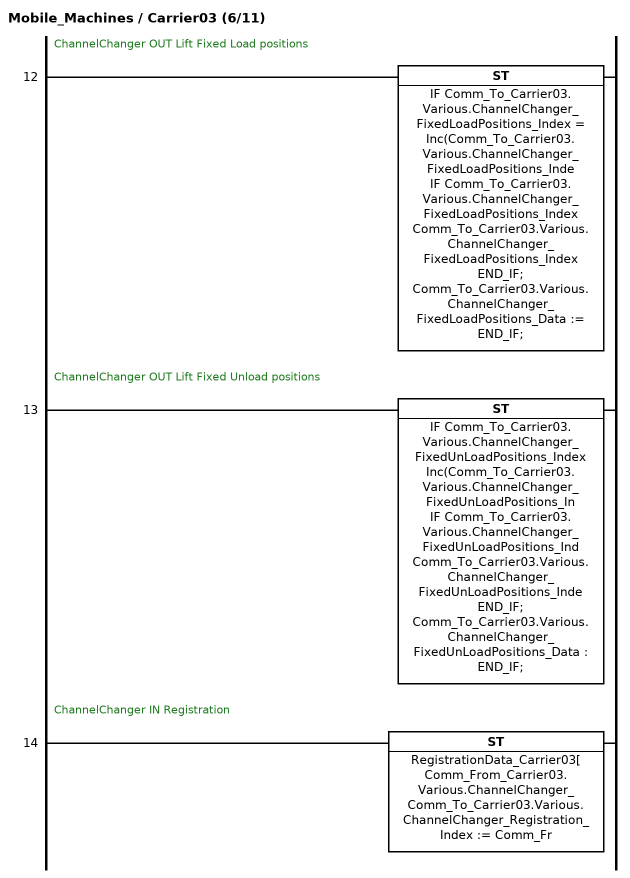
(* [picture p54: Mobile_Machines / Carrier03, rungs 12-14] *)
(* Rung 12: ChannelChanger OUT Lift Fixed Load positions *)
IF Comm_To_Carrier03.Various.ChannelChanger_FixedLoadPositions_Index = Comm_From_Carrier03.Various.ChannelChanger_FixedLoadPositions_Index THEN
	Inc(Comm_To_Carrier03.Various.ChannelChanger_FixedLoadPositions_Index);
	IF Comm_To_Carrier03.Various.ChannelChanger_FixedLoadPositions_Index > 199 THEN
		Comm_To_Carrier03.Various.ChannelChanger_FixedLoadPositions_Index := 0;
	END_IF;
	Comm_To_Carrier03.Various.ChannelChanger_FixedLoadPositions_Data := FixedLoadPosition_Array[Comm_To_Carrier03.Various.ChannelChanger_FixedLoadPositions_Index];
END_IF;
(* Rung 13: ChannelChanger OUT Lift Fixed Unload positions *)
IF Comm_To_Carrier03.Various.ChannelChanger_FixedUnLoadPositions_Index = Comm_From_Carrier03.Various.ChannelChanger_FixedUnLoadPositions_Index THEN
	Inc(Comm_To_Carrier03.Various.ChannelChanger_FixedUnLoadPositions_Index);
	IF Comm_To_Carrier03.Various.ChannelChanger_FixedUnLoadPositions_Index > 199 THEN
		Comm_To_Carrier03.Various.ChannelChanger_FixedUnLoadPositions_Index := 0;
	END_IF;
	Comm_To_Carrier03.Various.ChannelChanger_FixedUnLoadPositions_Data := FixedUnloadPosition_Array[Comm_To_Carrier03.Various.ChannelChanger_FixedUnLoadPositions_Index];
END_IF;
(* Rung 14: ChannelChanger IN Registration *)
RegistrationData_Carrier03[Comm_From_Carrier03.Various.ChannelChanger_Registration_Index] := Comm_From_Carrier03.Various.ChannelChanger_Registration_Data;
Comm_To_Carrier03.Various.ChannelChanger_Registration_Index := Comm_From_Carrier03.Various.ChannelChanger_Registration_Index;

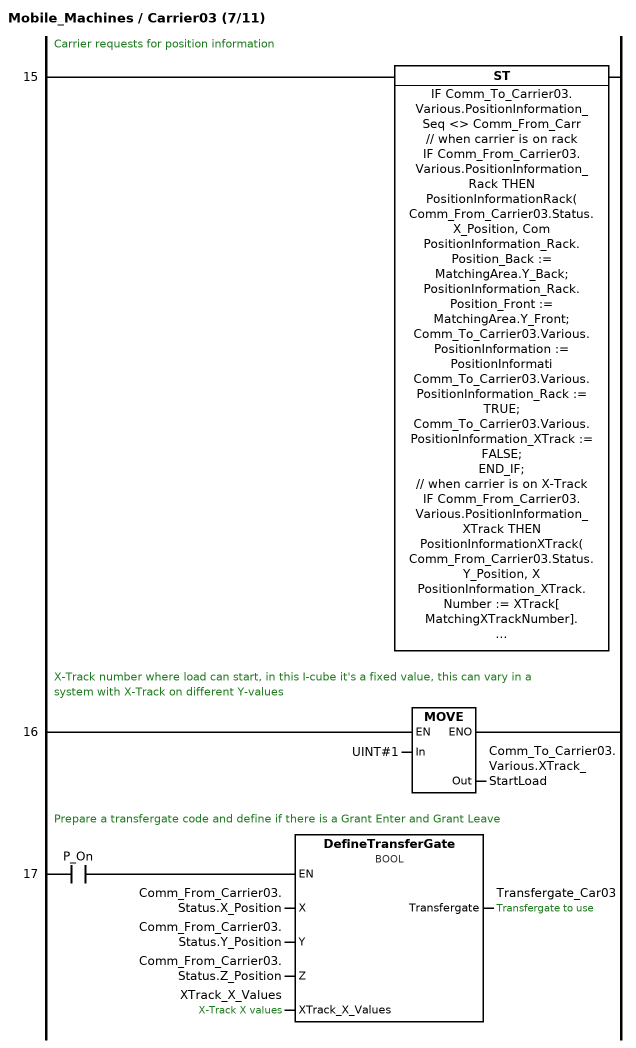
(* Rung 15: Carrier requests for position information *)
IF Comm_To_Carrier03.Various.PositionInformation_Seq <> Comm_From_Carrier03.Various.PositionInformation_Seq THEN
	// when carrier is on rack
	IF Comm_From_Carrier03.Various.PositionInformation_Rack THEN
		PositionInformationRack(Comm_From_Carrier03.Status.X_Position, Comm_From_Carrier03.Status.Y_Position, Comm_From_Carrier03.Status.Z_Position, Settings_CP.Margin_AreaCompare, Area, MatchingArea);
		PositionInformation_Rack.Position_Back := MatchingArea.Y_Back;
		PositionInformation_Rack.Position_Front := MatchingArea.Y_Front;
		Comm_To_Carrier03.Various.PositionInformation := PositionInformation_Rough;
		Comm_To_Carrier03.Various.PositionInformation_Rack := TRUE;
		Comm_To_Carrier03.Various.PositionInformation_XTrack := FALSE;
	END_IF;
	
	// when carrier is on X-Track
	IF Comm_From_Carrier03.Various.PositionInformation_XTrack THEN
		PositionInformationXTrack(Comm_From_Carrier03.Status.Y_Position, XTrack_Y_Values, MatchingXTrackNumber);
		PositionInformation_XTrack.Number := XTrack[MatchingXTrackNumber].XTrack_Number;
		PositionInformation_XTrack.Position_MIN := XTrack[MatchingXTrackNumber].MinimumPosition;
		PositionInformation_XTrack.Position_MAX := XTrack[MatchingXTrackNumber].MaximumPosition;
		Comm_To_Carrier03.Various.PositionInformation := PositionInformation_Rough;
		Comm_To_Carrier03.Various.PositionInformation_Rack := FALSE;
		Comm_To_Carrier03.Various.PositionInformation_XTrack := TRUE;
	END_IF;
	
	Comm_To_Carrier03.Various.PositionInformation_Seq := Comm_From_Carrier03.Various.PositionInformation_Seq;
	
END_IF;
(* Rung 16: X-Track number where load can start, in this I-cube it's a fixed value, this can vary in a system with X-Track on different Y-values *)
Comm_To_Carrier03.Various.XTrack_StartLoad := UINT#1;
(* Rung 17: Prepare a transfergate code and define if there is a Grant Enter and Grant Leave *)
_t32 := FALSE;
IF P_On THEN _t32 := DefineTransferGate(X := Comm_From_Carrier03.Status.X_Position, Y := Comm_From_Carrier03.Status.Y_Position, Z := Comm_From_Carrier03.Status.Z_Position, XTrack_X_Values := XTrack_X_Values, Transfergate => Transfergate_Car03); END_IF;

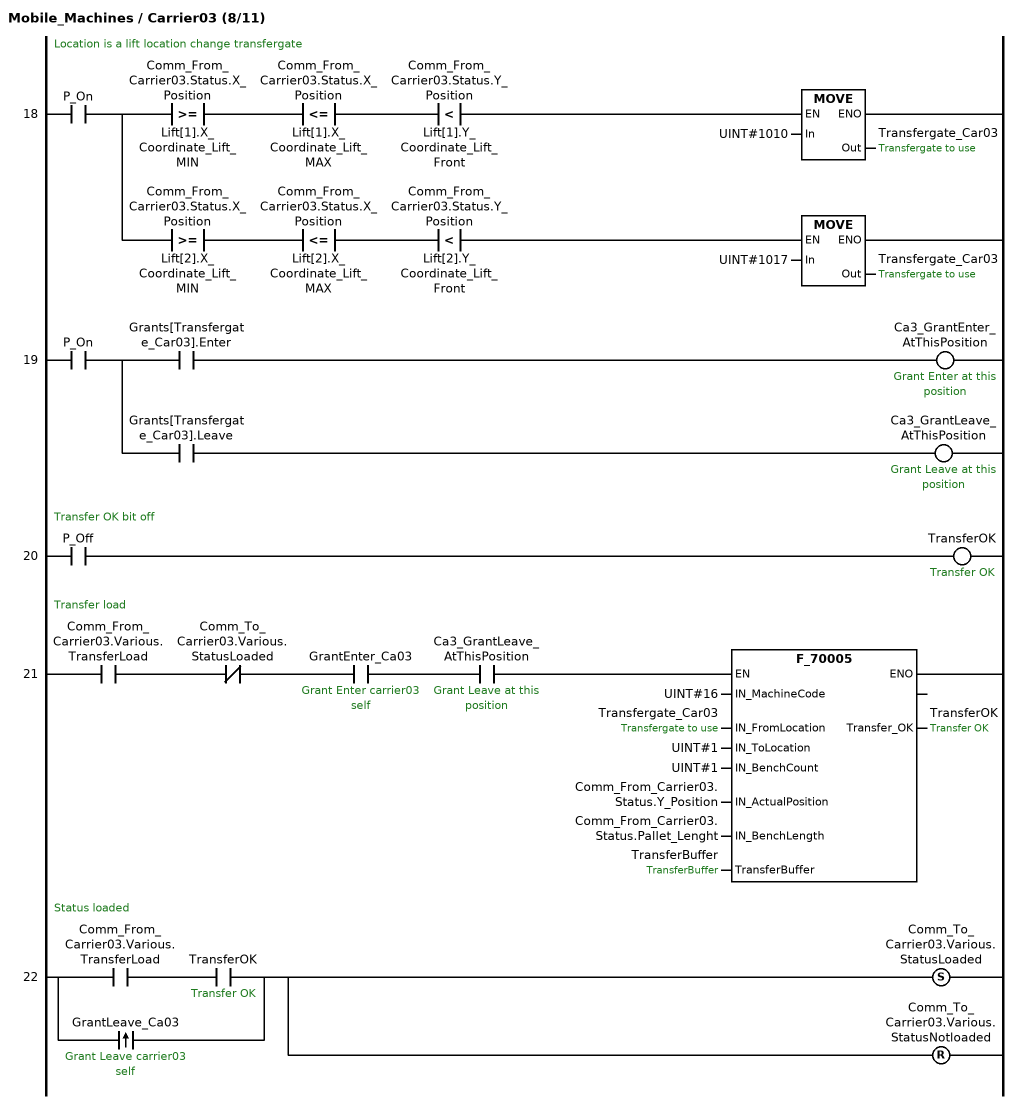
(* Rung 18: Location is a lift location change transfergate *)
IF P_On AND (Comm_From_Carrier03.Status.X_Position >= Lift[1].X_Coordinate_Lift_MIN) AND (Comm_From_Carrier03.Status.X_Position <= Lift[1].X_Coordinate_Lift_MAX) AND (Comm_From_Carrier03.Status.Y_Position < Lift[1].Y_Coordinate_Lift_Front) THEN
    Transfergate_Car03 := UINT#1010;
END_IF;
IF P_On AND (Comm_From_Carrier03.Status.X_Position >= Lift[2].X_Coordinate_Lift_MIN) AND (Comm_From_Carrier03.Status.X_Position <= Lift[2].X_Coordinate_Lift_MAX) AND (Comm_From_Carrier03.Status.Y_Position < Lift[2].Y_Coordinate_Lift_Front) THEN
    Transfergate_Car03 := UINT#1017;
END_IF;
(* Rung 19 *)
Ca3_GrantEnter_AtThisPosition := P_On AND Grants[Transfergate_Car03].Enter;
Ca3_GrantLeave_AtThisPosition := P_On AND Grants[Transfergate_Car03].Leave;
(* Rung 20: Transfer OK bit off *)
TransferOK := P_Off;
(* Rung 21: Transfer load *)
IF Comm_From_Carrier03.Various.TransferLoad AND NOT Comm_To_Carrier03.Various.StatusLoaded AND GrantEnter_Ca03 AND Ca3_GrantLeave_AtThisPosition THEN
    F_70005(IN_MachineCode := UINT#16, IN_FromLocation := Transfergate_Car03, IN_ToLocation := UINT#1, IN_BenchCount := UINT#1, IN_ActualPosition := Comm_From_Carrier03.Status.Y_Position, IN_BenchLength := Comm_From_Carrier03.Status.Pallet_Lenght, TransferBuffer := TransferBuffer, Transfer_OK => TransferOK);
END_IF;
(* Rung 22: Status loaded *)
_e33(CLK := GrantLeave_Ca03);
_p34 := (Comm_From_Carrier03.Various.TransferLoad AND TransferOK) OR _e33.Q;
IF _p34 THEN
    Comm_To_Carrier03.Various.StatusLoaded := TRUE;
    Comm_To_Carrier03.Various.StatusNotloaded := FALSE;
END_IF;

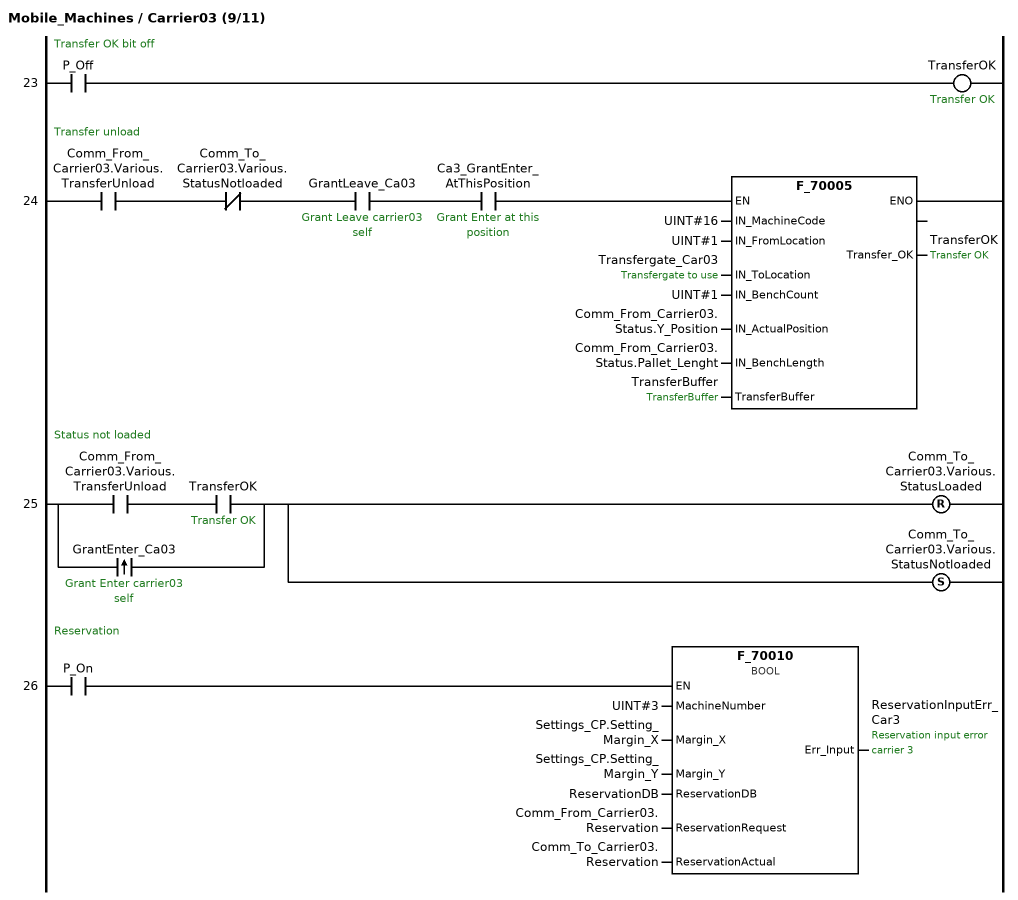
(* Rung 23: Transfer OK bit off *)
TransferOK := P_Off;
(* Rung 24: Transfer unload *)
IF Comm_From_Carrier03.Various.TransferUnload AND NOT Comm_To_Carrier03.Various.StatusNotloaded AND GrantLeave_Ca03 AND Ca3_GrantEnter_AtThisPosition THEN
    F_70005(IN_MachineCode := UINT#16, IN_FromLocation := UINT#1, IN_ToLocation := Transfergate_Car03, IN_BenchCount := UINT#1, IN_ActualPosition := Comm_From_Carrier03.Status.Y_Position, IN_BenchLength := Comm_From_Carrier03.Status.Pallet_Lenght, TransferBuffer := TransferBuffer, Transfer_OK => TransferOK);
END_IF;
(* Rung 25: Status not loaded *)
_e35(CLK := GrantEnter_Ca03);
_p36 := (Comm_From_Carrier03.Various.TransferUnload AND TransferOK) OR _e35.Q;
IF _p36 THEN
    Comm_To_Carrier03.Various.StatusLoaded := FALSE;
    Comm_To_Carrier03.Various.StatusNotloaded := TRUE;
END_IF;
(* Rung 26: Reservation *)
_t37 := FALSE;
IF P_On THEN _t37 := F_70010(MachineNumber := UINT#3, Margin_X := Settings_CP.Setting_Margin_X, Margin_Y := Settings_CP.Setting_Margin_Y, ReservationDB := ReservationDB, ReservationRequest := Comm_From_Carrier03.Reservation, ReservationActual := Comm_To_Carrier03.Reservation, Err_Input => ReservationInputErr_Car3); END_IF;

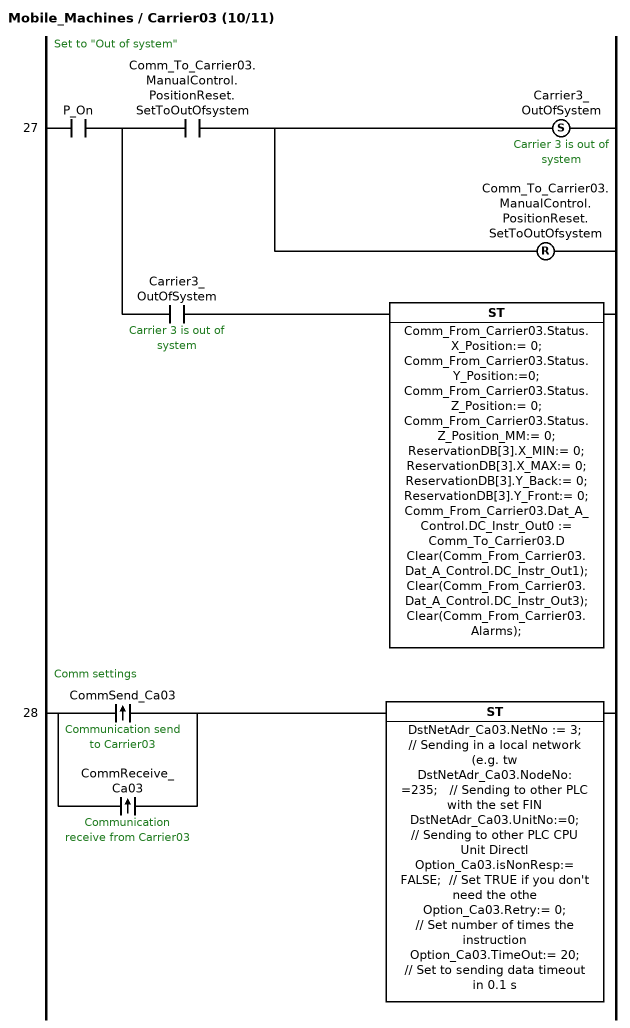
(* Rung 27: Set to "Out of system" *)
_p38 := P_On AND Comm_To_Carrier03.ManualControl.PositionReset.SetToOutOfsystem;
IF _p38 THEN
    Carrier3_OutOfSystem := TRUE;
    Comm_To_Carrier03.ManualControl.PositionReset.SetToOutOfsystem := FALSE;
END_IF;
IF P_On AND Carrier3_OutOfSystem THEN
    Comm_From_Carrier03.Status.X_Position:= 0;
    Comm_From_Carrier03.Status.Y_Position:=0;
    Comm_From_Carrier03.Status.Z_Position:= 0;
    Comm_From_Carrier03.Status.Z_Position_MM:= 0;
    
    ReservationDB[3].X_MIN:= 0;
    ReservationDB[3].X_MAX:= 0;
    ReservationDB[3].Y_Back:= 0;
    ReservationDB[3].Y_Front:= 0;
    
    Comm_From_Carrier03.Dat_A_Control.DC_Instr_Out0 := Comm_To_Carrier03.Dat_A_Control.Instr_Sequencenumber;
    Clear(Comm_From_Carrier03.Dat_A_Control.DC_Instr_Out1);
    Clear(Comm_From_Carrier03.Dat_A_Control.DC_Instr_Out3);
    Clear(Comm_From_Carrier03.Alarms);
END_IF;
(* Rung 28: Comm settings *)
_e39(CLK := CommSend_Ca03);
_e40(CLK := CommReceive_Ca03);
IF _e39.Q OR _e40.Q THEN
    DstNetAdr_Ca03.NetNo := 3;			// Sending in a local network (e.g. two PLCs connected by Ethernet LAN vai a hub)
    DstNetAdr_Ca03.NodeNo:=235;		// Sending to other PLC with the set FINS Node NUmber (depending on the other PLC)
    DstNetAdr_Ca03.UnitNo:=0;			// Sending to other PLC CPU Unit Directly
    
    Option_Ca03.isNonResp:= FALSE; 	// Set TRUE if you don't need the other CPU to reply back, otherwise set to FALSE
    Option_Ca03.Retry:= 0;					// Set number of times the instruction will retry sending if it failed to send data
    Option_Ca03.TimeOut:= 20;			// Set to sending data timeout in 0.1 s unit (e.g. 20 = 2 secs)
END_IF;

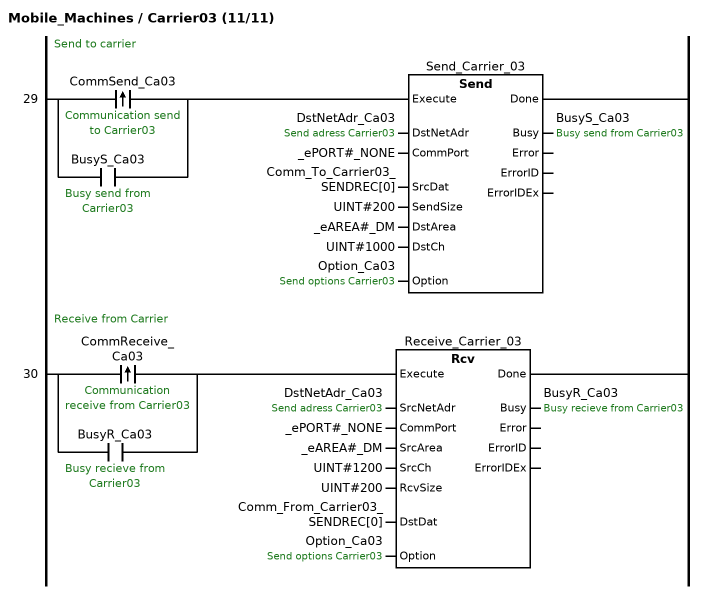
(* Rung 29: Send to carrier *)
_e41(CLK := CommSend_Ca03);
Send_Carrier_03(Execute := _e41.Q OR BusyS_Ca03, DstNetAdr := DstNetAdr_Ca03, CommPort := _ePORT#_NONE, SrcDat := Comm_To_Carrier03_SENDREC[0], SendSize := UINT#200, DstArea := _eAREA#_DM, DstCh := UINT#1000, Option := Option_Ca03, Busy => BusyS_Ca03);
(* Rung 30: Receive from Carrier *)
_e42(CLK := CommReceive_Ca03);
Receive_Carrier_03(Execute := _e42.Q OR BusyR_Ca03, SrcNetAdr := DstNetAdr_Ca03, CommPort := _ePORT#_NONE, SrcArea := _eAREA#_DM, SrcCh := UINT#1200, RcvSize := UINT#200, DstDat := Comm_From_Carrier03_SENDREC[0], Option := Option_Ca03, Busy => BusyR_Ca03);

(* Section Carrier04: ladder, written here as Structured Text *)

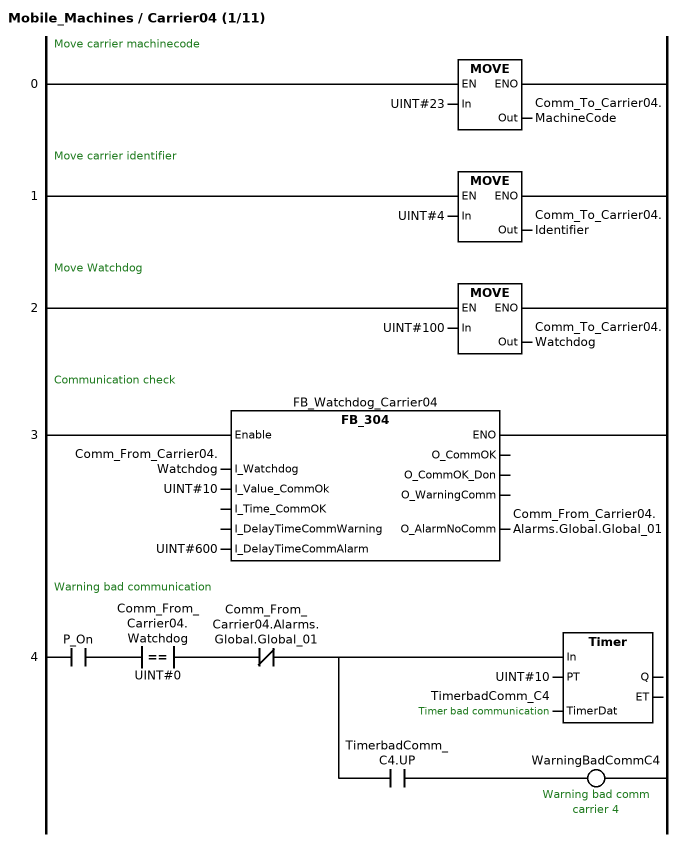
(* Rung 0: Move carrier machinecode *)
Comm_To_Carrier04.MachineCode := UINT#23;
(* Rung 1: Move carrier identifier *)
Comm_To_Carrier04.Identifier := UINT#4;
(* Rung 2: Move Watchdog *)
Comm_To_Carrier04.Watchdog := UINT#100;
(* Rung 3: Communication check *)
FB_Watchdog_Carrier04(Enable := TRUE, I_Watchdog := Comm_From_Carrier04.Watchdog, I_Value_CommOk := UINT#10, I_DelayTimeCommAlarm := UINT#600, O_AlarmNoComm => Comm_From_Carrier04.Alarms.Global.Global_01);
(* Rung 4: Warning bad communication *)
_p43 := P_On AND (Comm_From_Carrier04.Watchdog = UINT#0) AND NOT Comm_From_Carrier04.Alarms.Global.Global_01;
_t44 := Timer(In := _p43, PT := UINT#10, TimerDat := TimerbadComm_C4);
WarningBadCommC4 := _p43 AND TimerbadComm_C4.UP;

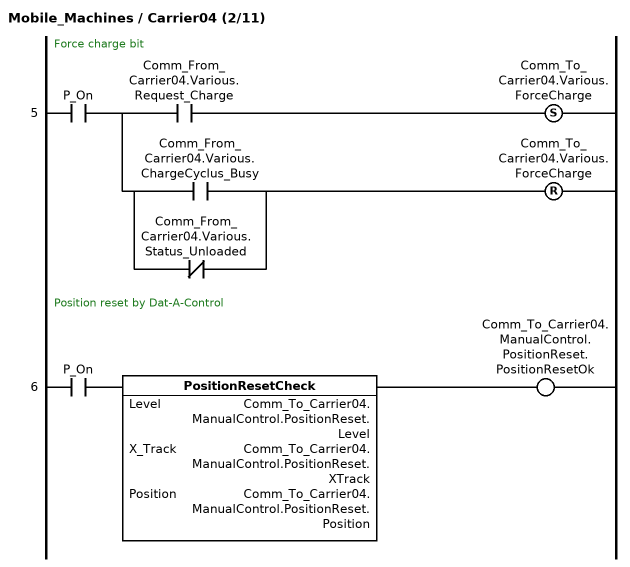
(* Rung 5: Force charge bit *)
IF P_On AND Comm_From_Carrier04.Various.Request_Charge THEN
    Comm_To_Carrier04.Various.ForceCharge := TRUE;
END_IF;
IF P_On AND (Comm_From_Carrier04.Various.ChargeCyclus_Busy OR NOT Comm_From_Carrier04.Various.Status_Unloaded) THEN
    Comm_To_Carrier04.Various.ForceCharge := FALSE;
END_IF;
(* Rung 6: Position reset by Dat-A-Control *)
Comm_To_Carrier04.ManualControl.PositionReset.PositionResetOk := P_On AND PositionResetCheck(Level := Comm_To_Carrier04.ManualControl.PositionReset.Level, X_Track := Comm_To_Carrier04.ManualControl.PositionReset.XTrack, Position := Comm_To_Carrier04.ManualControl.PositionReset.Position);

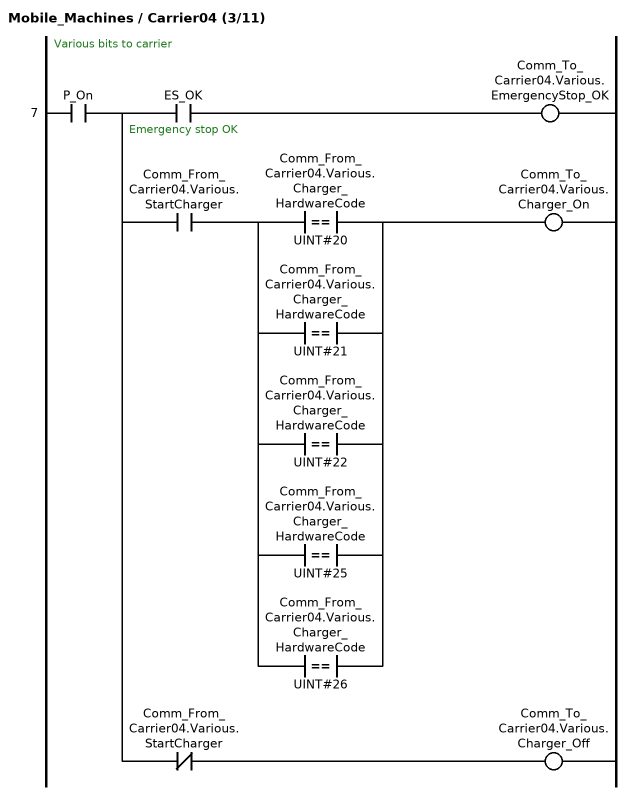
(* Rung 7: Various bits to carrier *)
Comm_To_Carrier04.Various.EmergencyStop_OK := P_On AND ES_OK;
Comm_To_Carrier04.Various.Charger_On := P_On AND Comm_From_Carrier04.Various.StartCharger AND ((Comm_From_Carrier04.Various.Charger_HardwareCode = UINT#20) OR (Comm_From_Carrier04.Various.Charger_HardwareCode = UINT#21) OR (Comm_From_Carrier04.Various.Charger_HardwareCode = UINT#22) OR (Comm_From_Carrier04.Various.Charger_HardwareCode = UINT#25) OR (Comm_From_Carrier04.Various.Charger_HardwareCode = UINT#26));
Comm_To_Carrier04.Various.Charger_Off := P_On AND NOT Comm_From_Carrier04.Various.StartCharger;

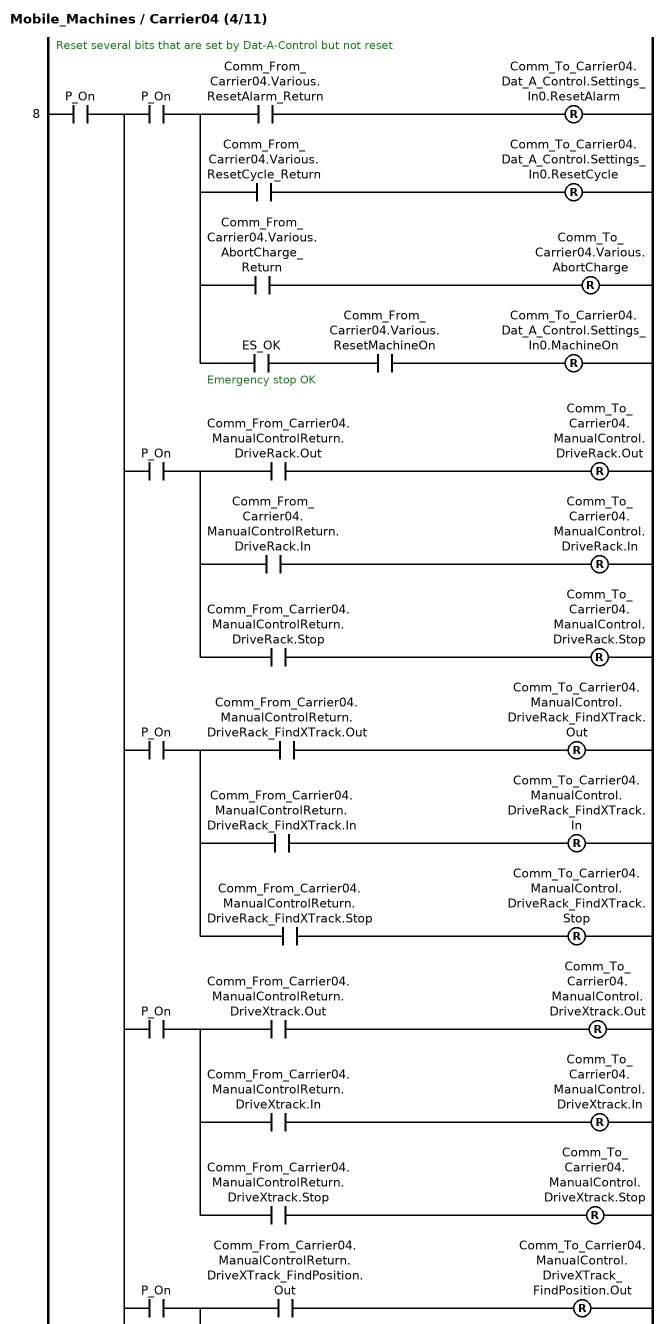

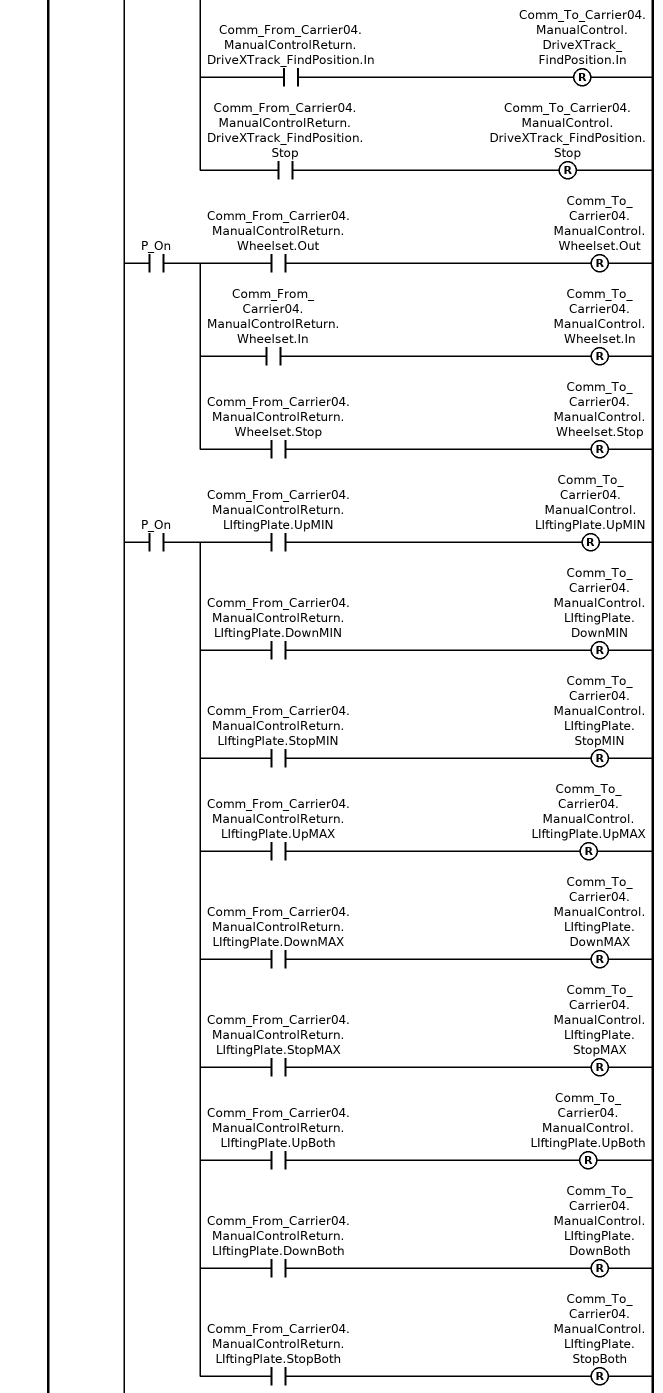

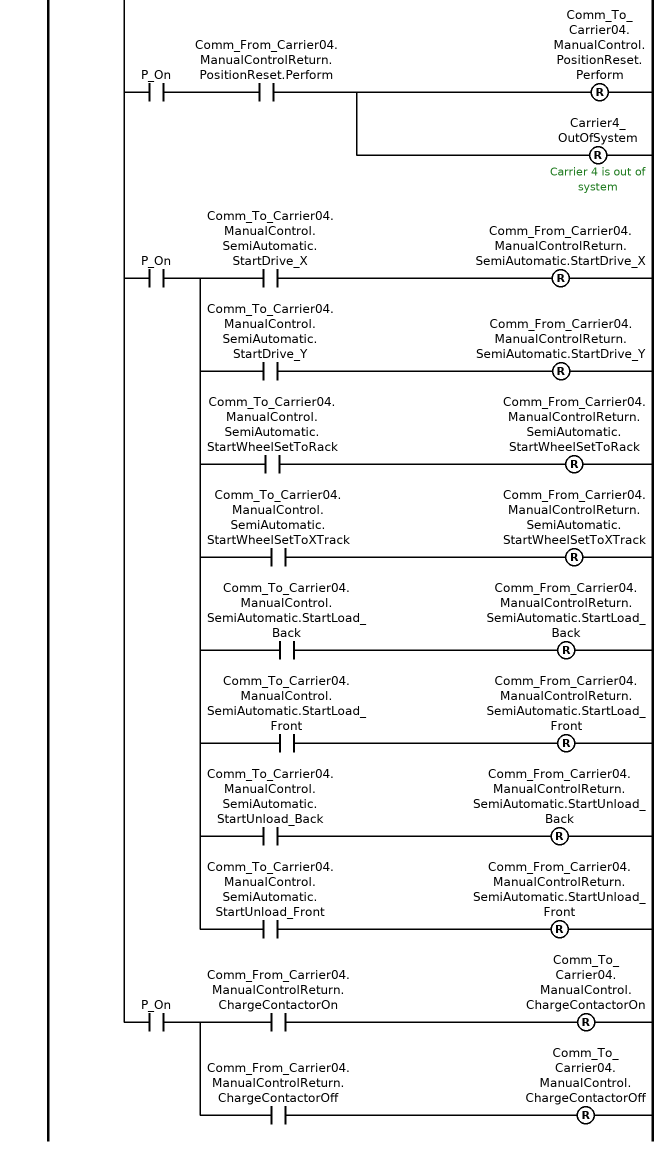
(* Rung 8: Reset several bits that are set by Dat-A-Control but not reset *)
IF P_On AND P_On AND Comm_From_Carrier04.Various.ResetAlarm_Return THEN
    Comm_To_Carrier04.Dat_A_Control.Settings_In0.ResetAlarm := FALSE;
END_IF;
IF P_On AND P_On AND Comm_From_Carrier04.Various.ResetCycle_Return THEN
    Comm_To_Carrier04.Dat_A_Control.Settings_In0.ResetCycle := FALSE;
END_IF;
IF P_On AND P_On AND Comm_From_Carrier04.Various.AbortCharge_Return THEN
    Comm_To_Carrier04.Various.AbortCharge := FALSE;
END_IF;
IF P_On AND P_On AND ES_OK AND Comm_From_Carrier04.Various.ResetMachineOn THEN
    Comm_To_Carrier04.Dat_A_Control.Settings_In0.MachineOn := FALSE;
END_IF;
IF P_On AND P_On AND Comm_From_Carrier04.ManualControlReturn.DriveRack.Out THEN
    Comm_To_Carrier04.ManualControl.DriveRack.Out := FALSE;
END_IF;
IF P_On AND P_On AND Comm_From_Carrier04.ManualControlReturn.DriveRack.In THEN
    Comm_To_Carrier04.ManualControl.DriveRack.In := FALSE;
END_IF;
IF P_On AND P_On AND Comm_From_Carrier04.ManualControlReturn.DriveRack.Stop THEN
    Comm_To_Carrier04.ManualControl.DriveRack.Stop := FALSE;
END_IF;
IF P_On AND P_On AND Comm_From_Carrier04.ManualControlReturn.DriveRack_FindXTrack.Out THEN
    Comm_To_Carrier04.ManualControl.DriveRack_FindXTrack.Out := FALSE;
END_IF;
IF P_On AND P_On AND Comm_From_Carrier04.ManualControlReturn.DriveRack_FindXTrack.In THEN
    Comm_To_Carrier04.ManualControl.DriveRack_FindXTrack.In := FALSE;
END_IF;
IF P_On AND P_On AND Comm_From_Carrier04.ManualControlReturn.DriveRack_FindXTrack.Stop THEN
    Comm_To_Carrier04.ManualControl.DriveRack_FindXTrack.Stop := FALSE;
END_IF;
IF P_On AND P_On AND Comm_From_Carrier04.ManualControlReturn.DriveXtrack.Out THEN
    Comm_To_Carrier04.ManualControl.DriveXtrack.Out := FALSE;
END_IF;
IF P_On AND P_On AND Comm_From_Carrier04.ManualControlReturn.DriveXtrack.In THEN
    Comm_To_Carrier04.ManualControl.DriveXtrack.In := FALSE;
END_IF;
IF P_On AND P_On AND Comm_From_Carrier04.ManualControlReturn.DriveXtrack.Stop THEN
    Comm_To_Carrier04.ManualControl.DriveXtrack.Stop := FALSE;
END_IF;
IF P_On AND P_On AND Comm_From_Carrier04.ManualControlReturn.DriveXTrack_FindPosition.Out THEN
    Comm_To_Carrier04.ManualControl.DriveXTrack_FindPosition.Out := FALSE;
END_IF;
IF P_On AND P_On AND Comm_From_Carrier04.ManualControlReturn.DriveXTrack_FindPosition.In THEN
    Comm_To_Carrier04.ManualControl.DriveXTrack_FindPosition.In := FALSE;
END_IF;
IF P_On AND P_On AND Comm_From_Carrier04.ManualControlReturn.DriveXTrack_FindPosition.Stop THEN
    Comm_To_Carrier04.ManualControl.DriveXTrack_FindPosition.Stop := FALSE;
END_IF;
IF P_On AND P_On AND Comm_From_Carrier04.ManualControlReturn.Wheelset.Out THEN
    Comm_To_Carrier04.ManualControl.Wheelset.Out := FALSE;
END_IF;
IF P_On AND P_On AND Comm_From_Carrier04.ManualControlReturn.Wheelset.In THEN
    Comm_To_Carrier04.ManualControl.Wheelset.In := FALSE;
END_IF;
IF P_On AND P_On AND Comm_From_Carrier04.ManualControlReturn.Wheelset.Stop THEN
    Comm_To_Carrier04.ManualControl.Wheelset.Stop := FALSE;
END_IF;
IF P_On AND P_On AND Comm_From_Carrier04.ManualControlReturn.LIftingPlate.UpMIN THEN
    Comm_To_Carrier04.ManualControl.LIftingPlate.UpMIN := FALSE;
END_IF;
IF P_On AND P_On AND Comm_From_Carrier04.ManualControlReturn.LIftingPlate.DownMIN THEN
    Comm_To_Carrier04.ManualControl.LIftingPlate.DownMIN := FALSE;
END_IF;
IF P_On AND P_On AND Comm_From_Carrier04.ManualControlReturn.LIftingPlate.StopMIN THEN
    Comm_To_Carrier04.ManualControl.LIftingPlate.StopMIN := FALSE;
END_IF;
IF P_On AND P_On AND Comm_From_Carrier04.ManualControlReturn.LIftingPlate.UpMAX THEN
    Comm_To_Carrier04.ManualControl.LIftingPlate.UpMAX := FALSE;
END_IF;
IF P_On AND P_On AND Comm_From_Carrier04.ManualControlReturn.LIftingPlate.DownMAX THEN
    Comm_To_Carrier04.ManualControl.LIftingPlate.DownMAX := FALSE;
END_IF;
IF P_On AND P_On AND Comm_From_Carrier04.ManualControlReturn.LIftingPlate.StopMAX THEN
    Comm_To_Carrier04.ManualControl.LIftingPlate.StopMAX := FALSE;
END_IF;
IF P_On AND P_On AND Comm_From_Carrier04.ManualControlReturn.LIftingPlate.UpBoth THEN
    Comm_To_Carrier04.ManualControl.LIftingPlate.UpBoth := FALSE;
END_IF;
IF P_On AND P_On AND Comm_From_Carrier04.ManualControlReturn.LIftingPlate.DownBoth THEN
    Comm_To_Carrier04.ManualControl.LIftingPlate.DownBoth := FALSE;
END_IF;
IF P_On AND P_On AND Comm_From_Carrier04.ManualControlReturn.LIftingPlate.StopBoth THEN
    Comm_To_Carrier04.ManualControl.LIftingPlate.StopBoth := FALSE;
END_IF;
_p45 := P_On AND P_On AND Comm_From_Carrier04.ManualControlReturn.PositionReset.Perform;
IF _p45 THEN
    Comm_To_Carrier04.ManualControl.PositionReset.Perform := FALSE;
    Carrier4_OutOfSystem := FALSE;
END_IF;
IF P_On AND P_On AND Comm_To_Carrier04.ManualControl.SemiAutomatic.StartDrive_X THEN
    Comm_From_Carrier04.ManualControlReturn.SemiAutomatic.StartDrive_X := FALSE;
END_IF;
IF P_On AND P_On AND Comm_To_Carrier04.ManualControl.SemiAutomatic.StartDrive_Y THEN
    Comm_From_Carrier04.ManualControlReturn.SemiAutomatic.StartDrive_Y := FALSE;
END_IF;
IF P_On AND P_On AND Comm_To_Carrier04.ManualControl.SemiAutomatic.StartWheelSetToRack THEN
    Comm_From_Carrier04.ManualControlReturn.SemiAutomatic.StartWheelSetToRack := FALSE;
END_IF;
IF P_On AND P_On AND Comm_To_Carrier04.ManualControl.SemiAutomatic.StartWheelSetToXTrack THEN
    Comm_From_Carrier04.ManualControlReturn.SemiAutomatic.StartWheelSetToXTrack := FALSE;
END_IF;
IF P_On AND P_On AND Comm_To_Carrier04.ManualControl.SemiAutomatic.StartLoad_Back THEN
    Comm_From_Carrier04.ManualControlReturn.SemiAutomatic.StartLoad_Back := FALSE;
END_IF;
IF P_On AND P_On AND Comm_To_Carrier04.ManualControl.SemiAutomatic.StartLoad_Front THEN
    Comm_From_Carrier04.ManualControlReturn.SemiAutomatic.StartLoad_Front := FALSE;
END_IF;
IF P_On AND P_On AND Comm_To_Carrier04.ManualControl.SemiAutomatic.StartUnload_Back THEN
    Comm_From_Carrier04.ManualControlReturn.SemiAutomatic.StartUnload_Back := FALSE;
END_IF;
IF P_On AND P_On AND Comm_To_Carrier04.ManualControl.SemiAutomatic.StartUnload_Front THEN
    Comm_From_Carrier04.ManualControlReturn.SemiAutomatic.StartUnload_Front := FALSE;
END_IF;
IF P_On AND P_On AND Comm_From_Carrier04.ManualControlReturn.ChargeContactorOn THEN
    Comm_To_Carrier04.ManualControl.ChargeContactorOn := FALSE;
END_IF;
IF P_On AND P_On AND Comm_From_Carrier04.ManualControlReturn.ChargeContactorOff THEN
    Comm_To_Carrier04.ManualControl.ChargeContactorOff := FALSE;
END_IF;

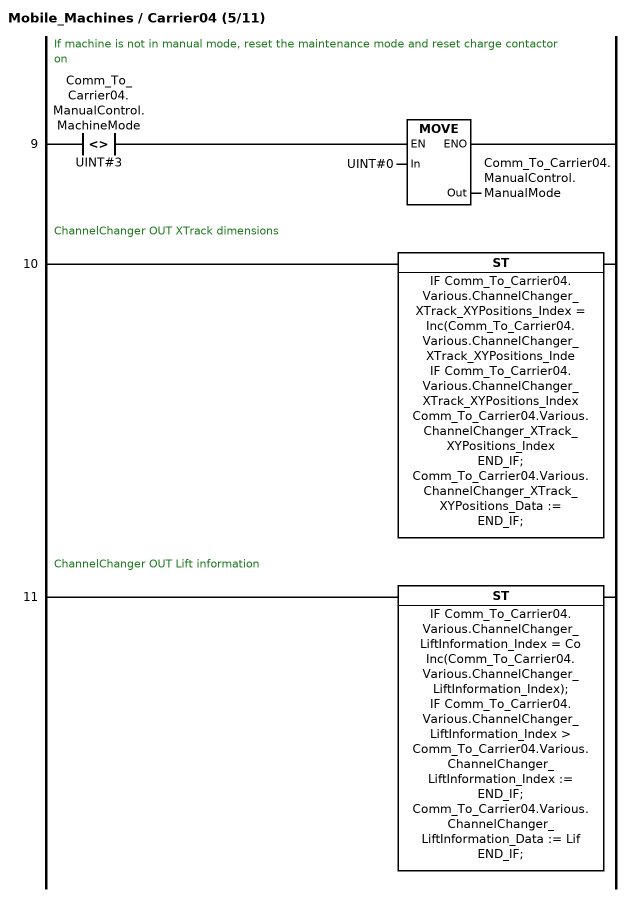
(* Rung 9: If machine is not in manual mode, reset the maintenance mode and reset charge contactor on *)
IF Comm_To_Carrier04.ManualControl.MachineMode <> UINT#3 THEN
    Comm_To_Carrier04.ManualControl.ManualMode := UINT#0;
END_IF;
(* Rung 10: ChannelChanger OUT XTrack dimensions *)
IF Comm_To_Carrier04.Various.ChannelChanger_XTrack_XYPositions_Index = Comm_From_Carrier04.Various.ChannelChanger_XTrack_XYPositions_Index THEN
	Inc(Comm_To_Carrier04.Various.ChannelChanger_XTrack_XYPositions_Index);
	IF Comm_To_Carrier04.Various.ChannelChanger_XTrack_XYPositions_Index > 199 THEN
		Comm_To_Carrier04.Various.ChannelChanger_XTrack_XYPositions_Index := 0;
	END_IF;
	Comm_To_Carrier04.Various.ChannelChanger_XTrack_XYPositions_Data := XTrack_XYPositions_Array[Comm_To_Carrier04.Various.ChannelChanger_XTrack_XYPositions_Index];
END_IF;
(* Rung 11: ChannelChanger OUT Lift information *)
IF Comm_To_Carrier04.Various.ChannelChanger_LiftInformation_Index = Comm_From_Carrier04.Various.ChannelChanger_LiftInformation_Index THEN
	Inc(Comm_To_Carrier04.Various.ChannelChanger_LiftInformation_Index);
	IF Comm_To_Carrier04.Various.ChannelChanger_LiftInformation_Index > 99 THEN
		Comm_To_Carrier04.Various.ChannelChanger_LiftInformation_Index := 0;
	END_IF;
	Comm_To_Carrier04.Various.ChannelChanger_LiftInformation_Data := Lift_Array[Comm_To_Carrier04.Various.ChannelChanger_LiftInformation_Index];
END_IF;

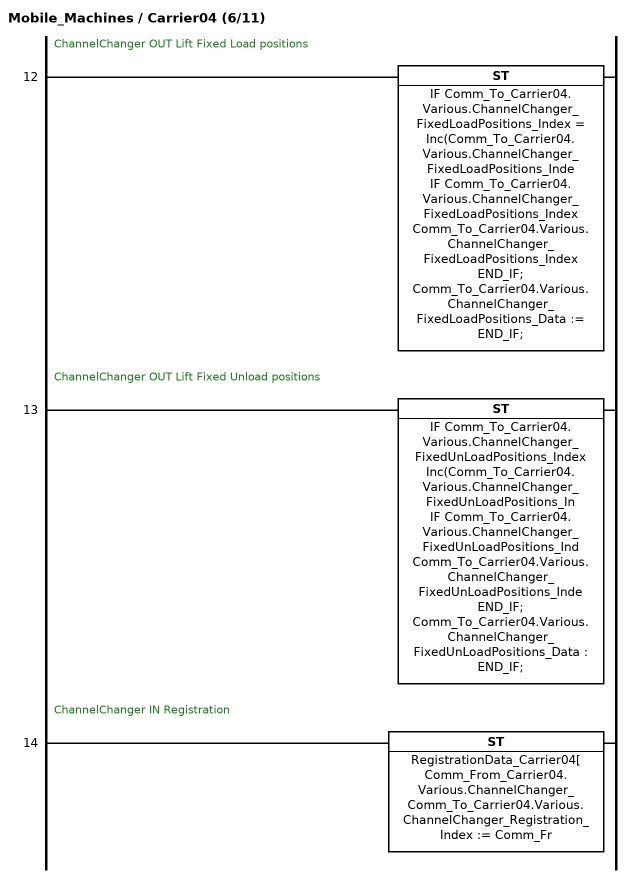
(* Rung 12: ChannelChanger OUT Lift Fixed Load positions *)
IF Comm_To_Carrier04.Various.ChannelChanger_FixedLoadPositions_Index = Comm_From_Carrier04.Various.ChannelChanger_FixedLoadPositions_Index THEN
	Inc(Comm_To_Carrier04.Various.ChannelChanger_FixedLoadPositions_Index);
	IF Comm_To_Carrier04.Various.ChannelChanger_FixedLoadPositions_Index > 199 THEN
		Comm_To_Carrier04.Various.ChannelChanger_FixedLoadPositions_Index := 0;
	END_IF;
	Comm_To_Carrier04.Various.ChannelChanger_FixedLoadPositions_Data := FixedLoadPosition_Array[Comm_To_Carrier04.Various.ChannelChanger_FixedLoadPositions_Index];
END_IF;
(* Rung 13: ChannelChanger OUT Lift Fixed Unload positions *)
IF Comm_To_Carrier04.Various.ChannelChanger_FixedUnLoadPositions_Index = Comm_From_Carrier04.Various.ChannelChanger_FixedUnLoadPositions_Index THEN
	Inc(Comm_To_Carrier04.Various.ChannelChanger_FixedUnLoadPositions_Index);
	IF Comm_To_Carrier04.Various.ChannelChanger_FixedUnLoadPositions_Index > 199 THEN
		Comm_To_Carrier04.Various.ChannelChanger_FixedUnLoadPositions_Index := 0;
	END_IF;
	Comm_To_Carrier04.Various.ChannelChanger_FixedUnLoadPositions_Data := FixedUnloadPosition_Array[Comm_To_Carrier04.Various.ChannelChanger_FixedUnLoadPositions_Index];
END_IF;
(* Rung 14: ChannelChanger IN Registration *)
RegistrationData_Carrier04[Comm_From_Carrier04.Various.ChannelChanger_Registration_Index] := Comm_From_Carrier04.Various.ChannelChanger_Registration_Data;
Comm_To_Carrier04.Various.ChannelChanger_Registration_Index := Comm_From_Carrier04.Various.ChannelChanger_Registration_Index;

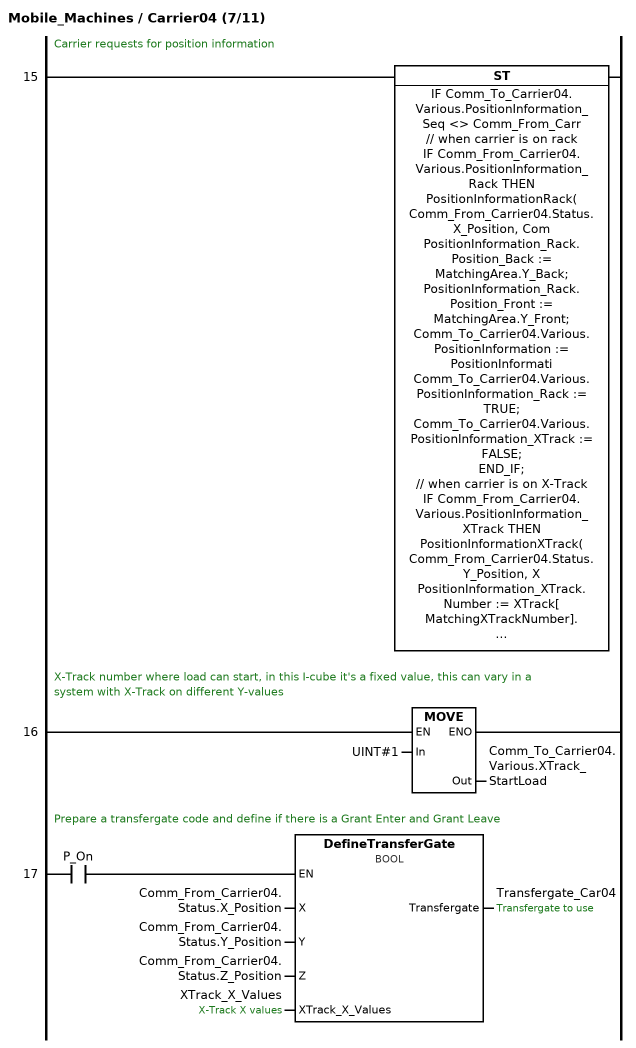
(* Rung 15: Carrier requests for position information *)
IF Comm_To_Carrier04.Various.PositionInformation_Seq <> Comm_From_Carrier04.Various.PositionInformation_Seq THEN
	// when carrier is on rack
	IF Comm_From_Carrier04.Various.PositionInformation_Rack THEN
		PositionInformationRack(Comm_From_Carrier04.Status.X_Position, Comm_From_Carrier04.Status.Y_Position, Comm_From_Carrier04.Status.Z_Position, Settings_CP.Margin_AreaCompare, Area, MatchingArea);
		PositionInformation_Rack.Position_Back := MatchingArea.Y_Back;
		PositionInformation_Rack.Position_Front := MatchingArea.Y_Front;
		Comm_To_Carrier04.Various.PositionInformation := PositionInformation_Rough;
		Comm_To_Carrier04.Various.PositionInformation_Rack := TRUE;
		Comm_To_Carrier04.Various.PositionInformation_XTrack := FALSE;
	END_IF;
	
	// when carrier is on X-Track
	IF Comm_From_Carrier04.Various.PositionInformation_XTrack THEN
		PositionInformationXTrack(Comm_From_Carrier04.Status.Y_Position, XTrack_Y_Values, MatchingXTrackNumber);
		PositionInformation_XTrack.Number := XTrack[MatchingXTrackNumber].XTrack_Number;
		PositionInformation_XTrack.Position_MIN := XTrack[MatchingXTrackNumber].MinimumPosition;
		PositionInformation_XTrack.Position_MAX := XTrack[MatchingXTrackNumber].MaximumPosition;
		Comm_To_Carrier04.Various.PositionInformation := PositionInformation_Rough;
		Comm_To_Carrier04.Various.PositionInformation_Rack := FALSE;
		Comm_To_Carrier04.Various.PositionInformation_XTrack := TRUE;
	END_IF;
	
	Comm_To_Carrier04.Various.PositionInformation_Seq := Comm_From_Carrier04.Various.PositionInformation_Seq;
	
END_IF;
(* Rung 16: X-Track number where load can start, in this I-cube it's a fixed value, this can vary in a system with X-Track on different Y-values *)
Comm_To_Carrier04.Various.XTrack_StartLoad := UINT#1;
(* Rung 17: Prepare a transfergate code and define if there is a Grant Enter and Grant Leave *)
_t46 := FALSE;
IF P_On THEN _t46 := DefineTransferGate(X := Comm_From_Carrier04.Status.X_Position, Y := Comm_From_Carrier04.Status.Y_Position, Z := Comm_From_Carrier04.Status.Z_Position, XTrack_X_Values := XTrack_X_Values, Transfergate => Transfergate_Car04); END_IF;

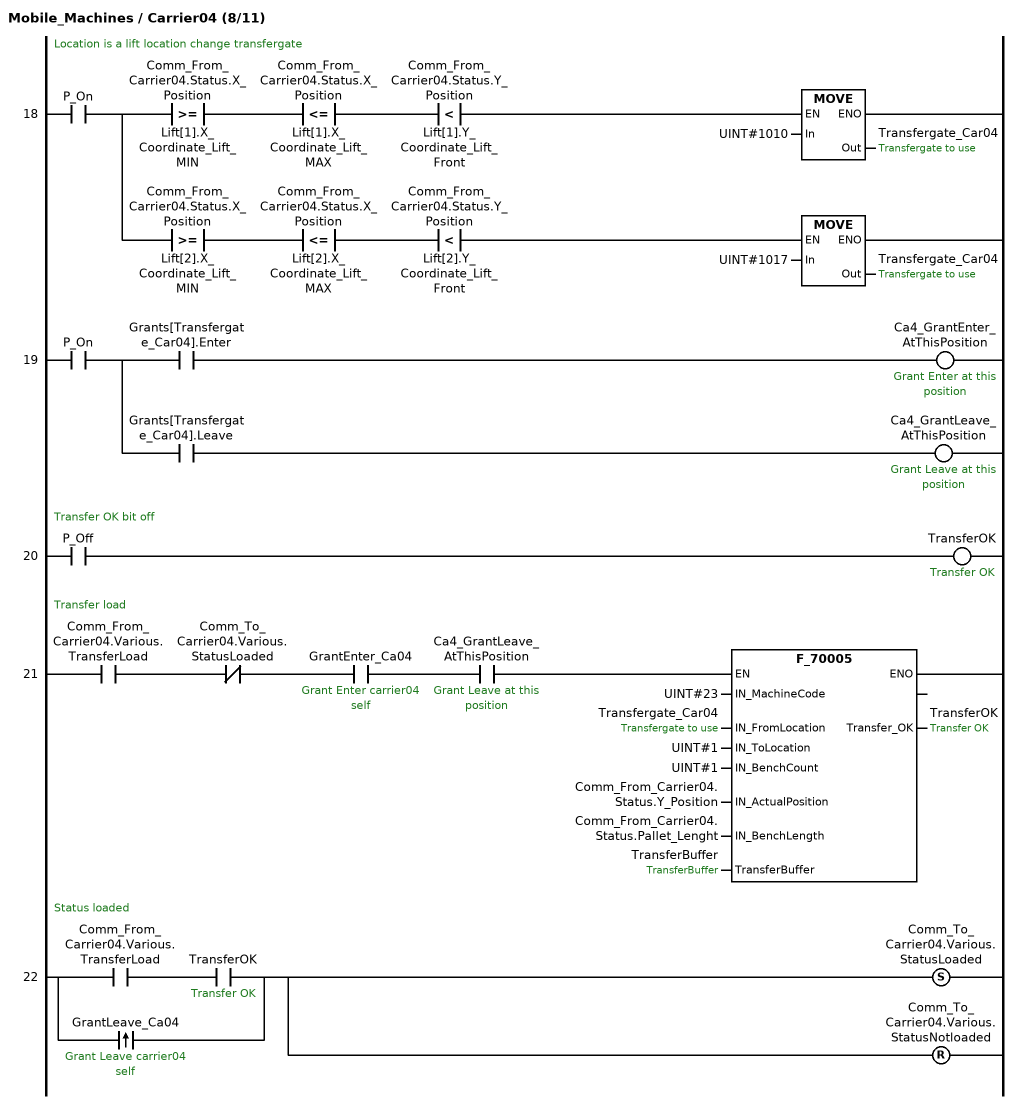
(* Rung 18: Location is a lift location change transfergate *)
IF P_On AND (Comm_From_Carrier04.Status.X_Position >= Lift[1].X_Coordinate_Lift_MIN) AND (Comm_From_Carrier04.Status.X_Position <= Lift[1].X_Coordinate_Lift_MAX) AND (Comm_From_Carrier04.Status.Y_Position < Lift[1].Y_Coordinate_Lift_Front) THEN
    Transfergate_Car04 := UINT#1010;
END_IF;
IF P_On AND (Comm_From_Carrier04.Status.X_Position >= Lift[2].X_Coordinate_Lift_MIN) AND (Comm_From_Carrier04.Status.X_Position <= Lift[2].X_Coordinate_Lift_MAX) AND (Comm_From_Carrier04.Status.Y_Position < Lift[2].Y_Coordinate_Lift_Front) THEN
    Transfergate_Car04 := UINT#1017;
END_IF;
(* Rung 19 *)
Ca4_GrantEnter_AtThisPosition := P_On AND Grants[Transfergate_Car04].Enter;
Ca4_GrantLeave_AtThisPosition := P_On AND Grants[Transfergate_Car04].Leave;
(* Rung 20: Transfer OK bit off *)
TransferOK := P_Off;
(* Rung 21: Transfer load *)
IF Comm_From_Carrier04.Various.TransferLoad AND NOT Comm_To_Carrier04.Various.StatusLoaded AND GrantEnter_Ca04 AND Ca4_GrantLeave_AtThisPosition THEN
    F_70005(IN_MachineCode := UINT#23, IN_FromLocation := Transfergate_Car04, IN_ToLocation := UINT#1, IN_BenchCount := UINT#1, IN_ActualPosition := Comm_From_Carrier04.Status.Y_Position, IN_BenchLength := Comm_From_Carrier04.Status.Pallet_Lenght, TransferBuffer := TransferBuffer, Transfer_OK => TransferOK);
END_IF;
(* Rung 22: Status loaded *)
_e47(CLK := GrantLeave_Ca04);
_p48 := (Comm_From_Carrier04.Various.TransferLoad AND TransferOK) OR _e47.Q;
IF _p48 THEN
    Comm_To_Carrier04.Various.StatusLoaded := TRUE;
    Comm_To_Carrier04.Various.StatusNotloaded := FALSE;
END_IF;

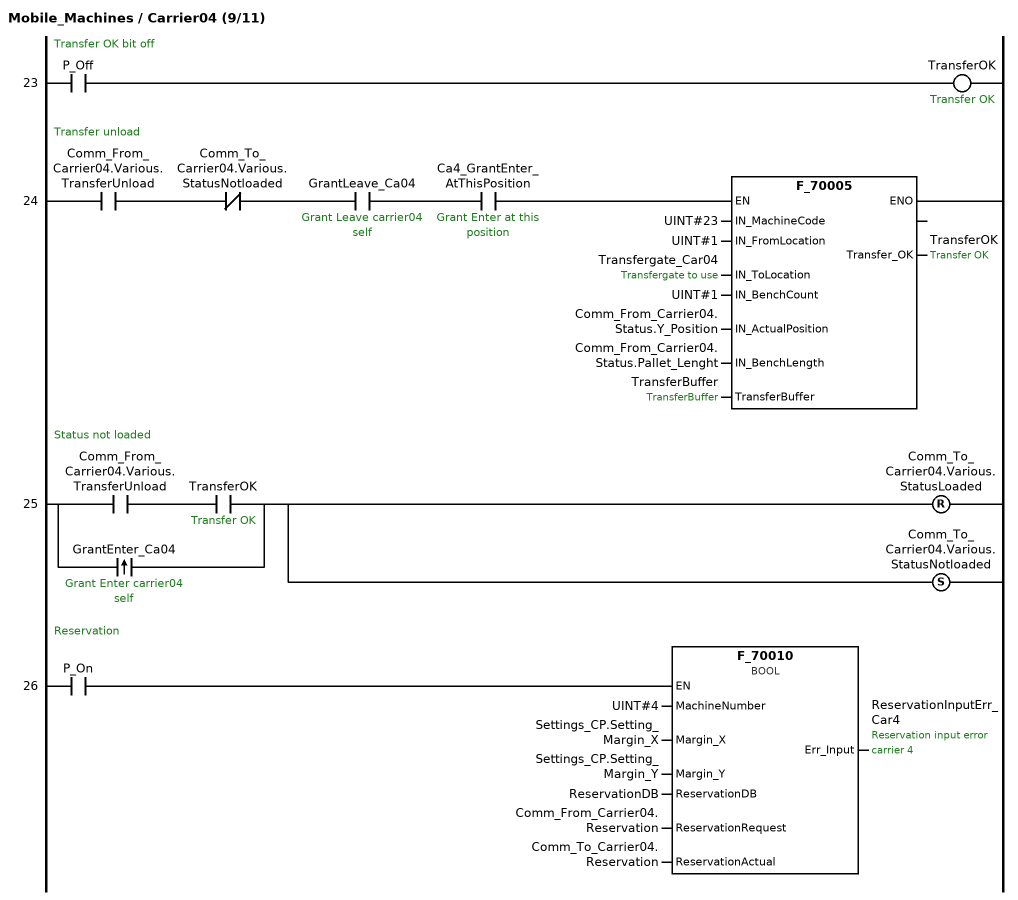
(* Rung 23: Transfer OK bit off *)
TransferOK := P_Off;
(* Rung 24: Transfer unload *)
IF Comm_From_Carrier04.Various.TransferUnload AND NOT Comm_To_Carrier04.Various.StatusNotloaded AND GrantLeave_Ca04 AND Ca4_GrantEnter_AtThisPosition THEN
    F_70005(IN_MachineCode := UINT#23, IN_FromLocation := UINT#1, IN_ToLocation := Transfergate_Car04, IN_BenchCount := UINT#1, IN_ActualPosition := Comm_From_Carrier04.Status.Y_Position, IN_BenchLength := Comm_From_Carrier04.Status.Pallet_Lenght, TransferBuffer := TransferBuffer, Transfer_OK => TransferOK);
END_IF;
(* Rung 25: Status not loaded *)
_e49(CLK := GrantEnter_Ca04);
_p50 := (Comm_From_Carrier04.Various.TransferUnload AND TransferOK) OR _e49.Q;
IF _p50 THEN
    Comm_To_Carrier04.Various.StatusLoaded := FALSE;
    Comm_To_Carrier04.Various.StatusNotloaded := TRUE;
END_IF;
(* Rung 26: Reservation *)
_t51 := FALSE;
IF P_On THEN _t51 := F_70010(MachineNumber := UINT#4, Margin_X := Settings_CP.Setting_Margin_X, Margin_Y := Settings_CP.Setting_Margin_Y, ReservationDB := ReservationDB, ReservationRequest := Comm_From_Carrier04.Reservation, ReservationActual := Comm_To_Carrier04.Reservation, Err_Input => ReservationInputErr_Car4); END_IF;

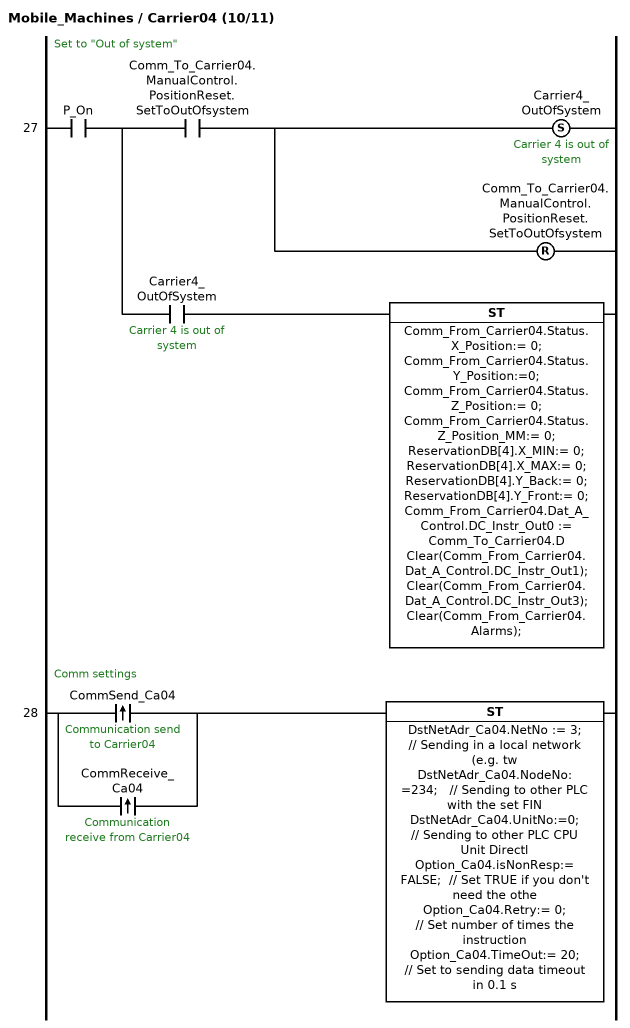
(* Rung 27: Set to "Out of system" *)
_p52 := P_On AND Comm_To_Carrier04.ManualControl.PositionReset.SetToOutOfsystem;
IF _p52 THEN
    Carrier4_OutOfSystem := TRUE;
    Comm_To_Carrier04.ManualControl.PositionReset.SetToOutOfsystem := FALSE;
END_IF;
IF P_On AND Carrier4_OutOfSystem THEN
    Comm_From_Carrier04.Status.X_Position:= 0;
    Comm_From_Carrier04.Status.Y_Position:=0;
    Comm_From_Carrier04.Status.Z_Position:= 0;
    Comm_From_Carrier04.Status.Z_Position_MM:= 0;
    
    ReservationDB[4].X_MIN:= 0;
    ReservationDB[4].X_MAX:= 0;
    ReservationDB[4].Y_Back:= 0;
    ReservationDB[4].Y_Front:= 0;
    
    Comm_From_Carrier04.Dat_A_Control.DC_Instr_Out0 := Comm_To_Carrier04.Dat_A_Control.Instr_Sequencenumber;
    Clear(Comm_From_Carrier04.Dat_A_Control.DC_Instr_Out1);
    Clear(Comm_From_Carrier04.Dat_A_Control.DC_Instr_Out3);
    Clear(Comm_From_Carrier04.Alarms);
END_IF;
(* Rung 28: Comm settings *)
_e53(CLK := CommSend_Ca04);
_e54(CLK := CommReceive_Ca04);
IF _e53.Q OR _e54.Q THEN
    DstNetAdr_Ca04.NetNo := 3;			// Sending in a local network (e.g. two PLCs connected by Ethernet LAN vai a hub)
    DstNetAdr_Ca04.NodeNo:=234;		// Sending to other PLC with the set FINS Node NUmber (depending on the other PLC)
    DstNetAdr_Ca04.UnitNo:=0;			// Sending to other PLC CPU Unit Directly
    
    Option_Ca04.isNonResp:= FALSE; 	// Set TRUE if you don't need the other CPU to reply back, otherwise set to FALSE
    Option_Ca04.Retry:= 0;					// Set number of times the instruction will retry sending if it failed to send data
    Option_Ca04.TimeOut:= 20;			// Set to sending data timeout in 0.1 s unit (e.g. 20 = 2 secs)
END_IF;

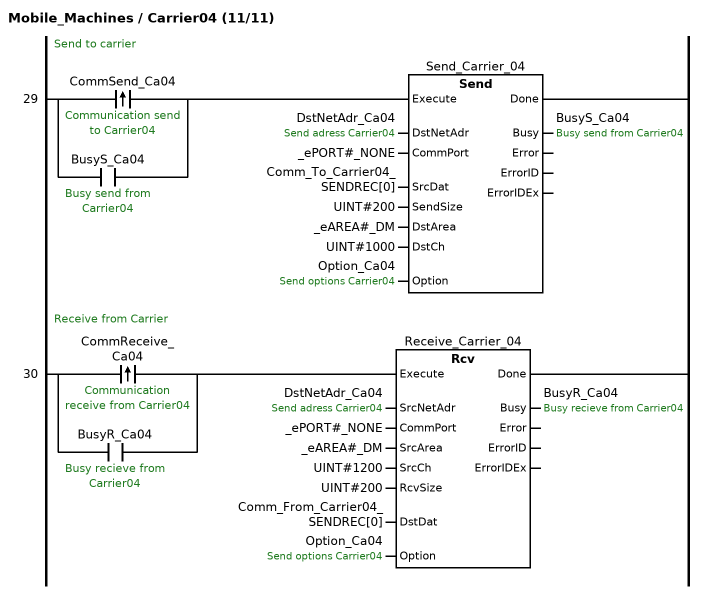
(* Rung 29: Send to carrier *)
_e55(CLK := CommSend_Ca04);
Send_Carrier_04(Execute := _e55.Q OR BusyS_Ca04, DstNetAdr := DstNetAdr_Ca04, CommPort := _ePORT#_NONE, SrcDat := Comm_To_Carrier04_SENDREC[0], SendSize := UINT#200, DstArea := _eAREA#_DM, DstCh := UINT#1000, Option := Option_Ca04, Busy => BusyS_Ca04);
(* Rung 30: Receive from Carrier *)
_e56(CLK := CommReceive_Ca04);
Receive_Carrier_04(Execute := _e56.Q OR BusyR_Ca04, SrcNetAdr := DstNetAdr_Ca04, CommPort := _ePORT#_NONE, SrcArea := _eAREA#_DM, SrcCh := UINT#1200, RcvSize := UINT#200, DstDat := Comm_From_Carrier04_SENDREC[0], Option := Option_Ca04, Busy => BusyR_Ca04);

(* Section Carrier05: ladder, written here as Structured Text *)

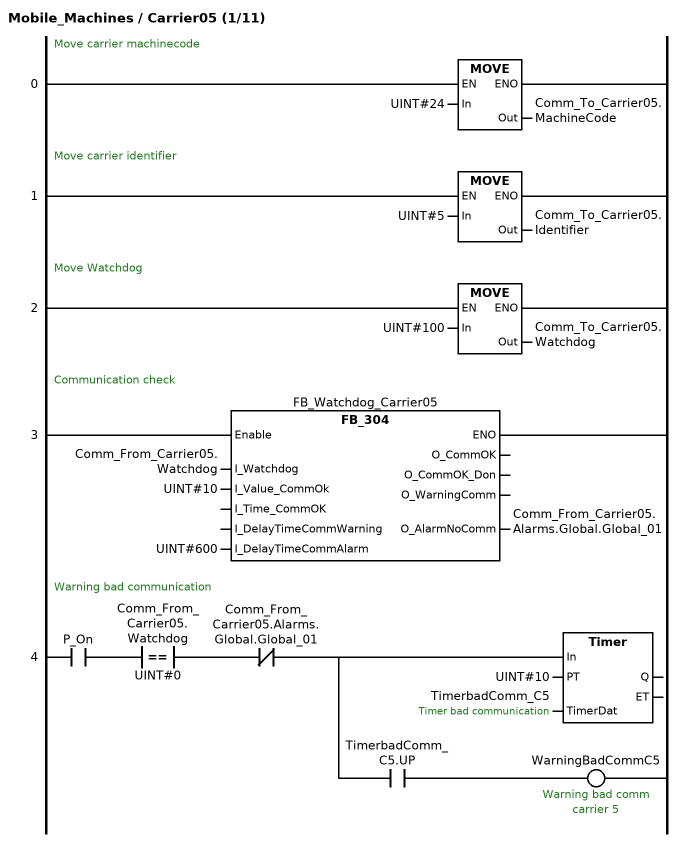
(* Rung 0: Move carrier machinecode *)
Comm_To_Carrier05.MachineCode := UINT#24;
(* Rung 1: Move carrier identifier *)
Comm_To_Carrier05.Identifier := UINT#5;
(* Rung 2: Move Watchdog *)
Comm_To_Carrier05.Watchdog := UINT#100;
(* Rung 3: Communication check *)
FB_Watchdog_Carrier05(Enable := TRUE, I_Watchdog := Comm_From_Carrier05.Watchdog, I_Value_CommOk := UINT#10, I_DelayTimeCommAlarm := UINT#600, O_AlarmNoComm => Comm_From_Carrier05.Alarms.Global.Global_01);
(* Rung 4: Warning bad communication *)
_p57 := P_On AND (Comm_From_Carrier05.Watchdog = UINT#0) AND NOT Comm_From_Carrier05.Alarms.Global.Global_01;
_t58 := Timer(In := _p57, PT := UINT#10, TimerDat := TimerbadComm_C5);
WarningBadCommC5 := _p57 AND TimerbadComm_C5.UP;

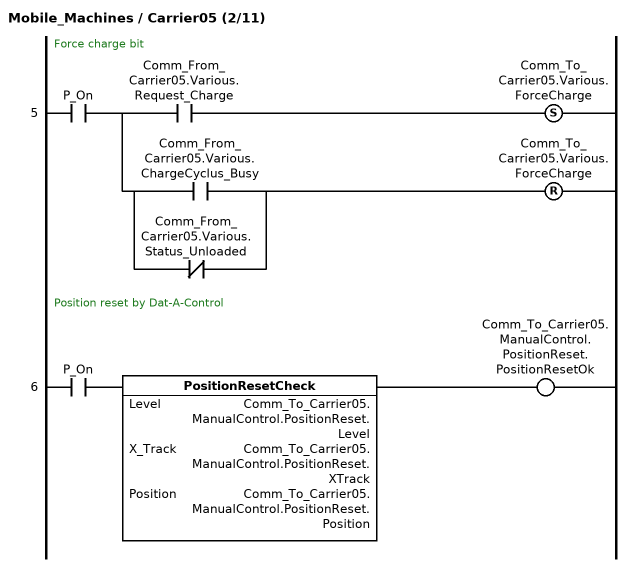
(* Rung 5: Force charge bit *)
IF P_On AND Comm_From_Carrier05.Various.Request_Charge THEN
    Comm_To_Carrier05.Various.ForceCharge := TRUE;
END_IF;
IF P_On AND (Comm_From_Carrier05.Various.ChargeCyclus_Busy OR NOT Comm_From_Carrier05.Various.Status_Unloaded) THEN
    Comm_To_Carrier05.Various.ForceCharge := FALSE;
END_IF;
(* Rung 6: Position reset by Dat-A-Control *)
Comm_To_Carrier05.ManualControl.PositionReset.PositionResetOk := P_On AND PositionResetCheck(Level := Comm_To_Carrier05.ManualControl.PositionReset.Level, X_Track := Comm_To_Carrier05.ManualControl.PositionReset.XTrack, Position := Comm_To_Carrier05.ManualControl.PositionReset.Position);

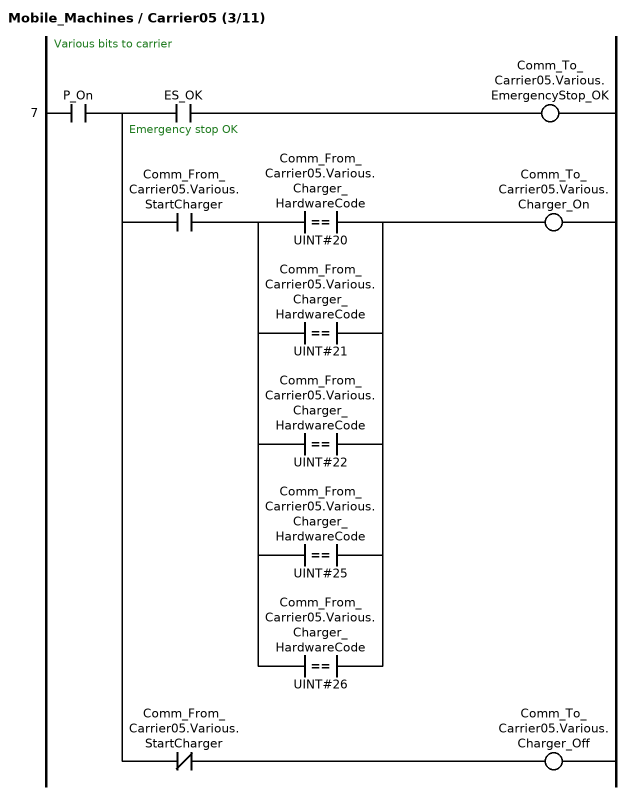
(* Rung 7: Various bits to carrier *)
Comm_To_Carrier05.Various.EmergencyStop_OK := P_On AND ES_OK;
Comm_To_Carrier05.Various.Charger_On := P_On AND Comm_From_Carrier05.Various.StartCharger AND ((Comm_From_Carrier05.Various.Charger_HardwareCode = UINT#20) OR (Comm_From_Carrier05.Various.Charger_HardwareCode = UINT#21) OR (Comm_From_Carrier05.Various.Charger_HardwareCode = UINT#22) OR (Comm_From_Carrier05.Various.Charger_HardwareCode = UINT#25) OR (Comm_From_Carrier05.Various.Charger_HardwareCode = UINT#26));
Comm_To_Carrier05.Various.Charger_Off := P_On AND NOT Comm_From_Carrier05.Various.StartCharger;

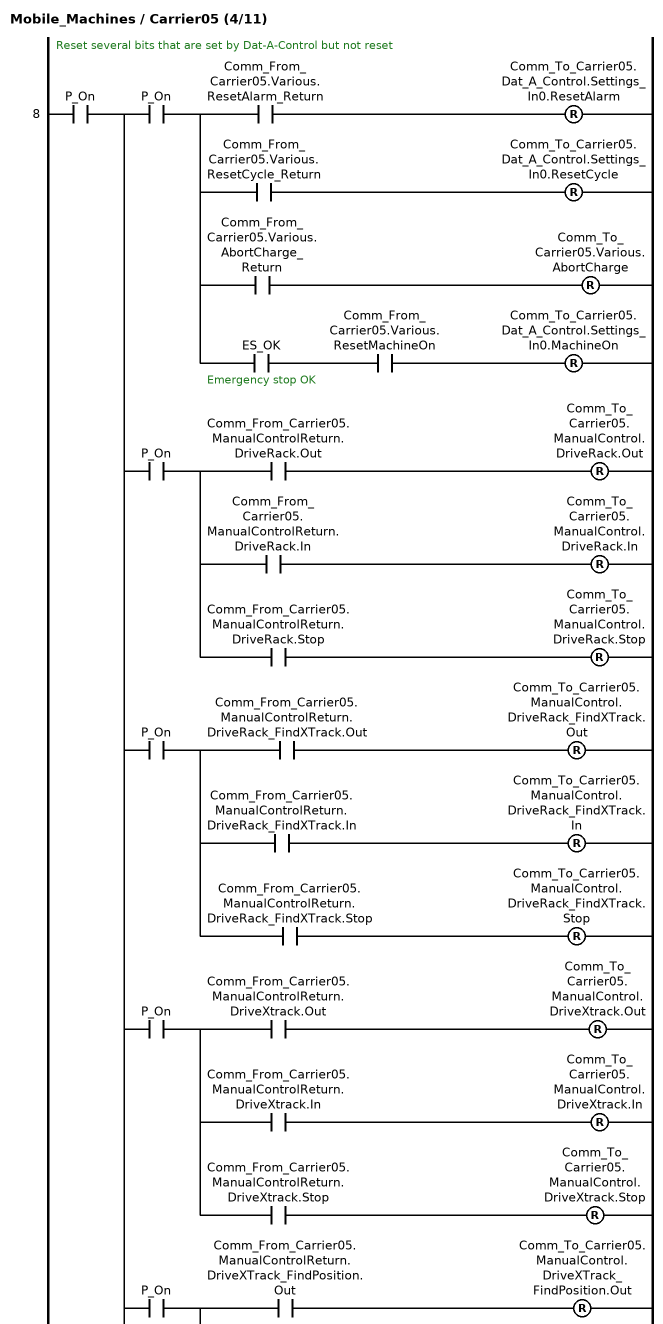

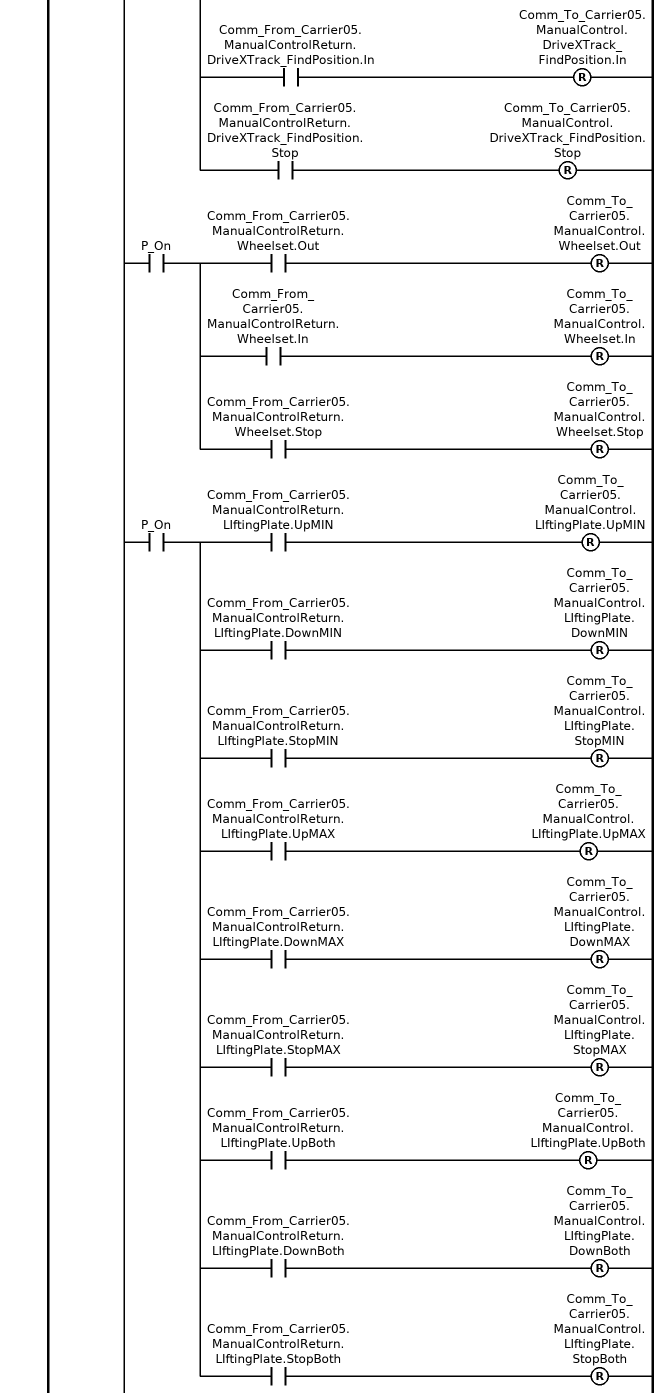

